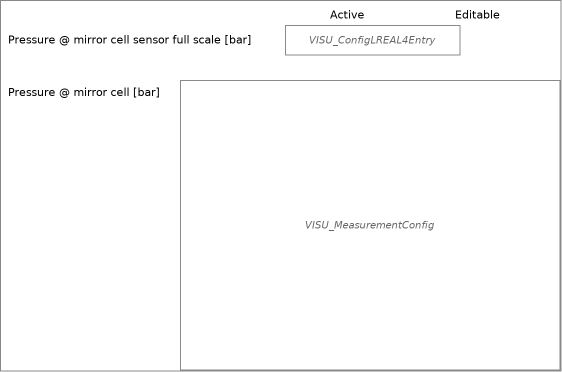
VISUALIZATION VISU_M1Config_Axial_MirrorPressure  // 562x372
VAR_IN_OUT
    editable : M1AxialSupportConfig;
	active : M1AxialSupportConfig;
END_VAR
    Label (285,5 125x20), "Active"
    Label (415,5 125x20), "Editable"
    Label (5,25 260x30), "Pressure @ mirror cell sensor full scale [bar]"
    Frame (285,25 175x30)
        shows VISU_ConfigLREAL4Entry(active := active.mirrorPressureSensorFullScale, editable := editable.mirrorPressureSensorFullScale)
    Label (5,60 170x65), "Pressure @ mirror cell [bar]"
    Frame (180,80 380x290)
        shows VISU_MeasurementConfig(active := active.mirrorPressure, editable := editable.mirrorPressure)
END_VISUALIZATION

(* stored: Version 1.1.0.1, ProductVersion 3.1.4019.2
   Visu VISU_M1Config_Axial_MirrorPressure: Id {7b9ca0a1-406c-4c7f-9e0f-06db3c022522} *)
